// TIA Portal V18 export
VAR_GLOBAL   // PLC tag table "FactoryIO"
   "Emergency Stop 0" AT %I0.0 : Bool;
   "Start Button 0" AT %I0.1 : Bool;
   "Stop Button 0" AT %I0.2 : Bool;
   "Reset Button 0" AT %I0.3 : Bool;
   "Machining Center 0 (Is Busy)" AT %I0.5 : Bool;
   "Machining Center 0 (Has Error)" AT %I0.6 : Bool;
   "Machining Center 1 (Is Busy)" AT %I0.7 : Bool;
   "Machining Center 1 (Has Error)" AT %I1.0 : Bool;
   "Sensor 120" AT %I1.1 : Bool;
   "Sensor 122" AT %I1.2 : Bool;
   "Zne01 Conveyor 101" AT %Q0.0 : Bool;
   "Zne01 Conveyor 120" AT %Q0.1 : Bool;
   "Zne01 Conveyor 121" AT %Q0.2 : Bool;
   "Zne01 Conveyor 122" AT %Q0.3 : Bool;
   "Zne01 Conveyor 124" AT %Q0.4 : Bool;
   "Zne01 Conveyor 125" AT %Q0.5 : Bool;
   "Zne01 Sorter 102 (Up)" AT %Q0.6 : Bool;
   "Zne01 Sorter 102 (Left)" AT %Q0.7 : Bool;
   "Zne01 Sorter 102 (Right)" AT %Q1.0 : Bool;
   "Zne01 Sorter 123 (Up)" AT %Q1.1 : Bool;
   "Zne01 Sorter 123 (Right)" AT %Q1.2 : Bool;
   "Machining Center 0 (Start)" AT %Q1.3 : Bool;
   "Machining Center 0 (Stop)" AT %Q1.4 : Bool;
   "Machining Center 0 (Reset)" AT %Q1.5 : Bool;
   "Machining Center 1 (Start)" AT %Q1.6 : Bool;
   "Machining Center 1 (Stop)" AT %Q1.7 : Bool;
   "Machining Center 1 (Reset)" AT %Q2.0 : Bool;
   "Start Button 0 (Light)" AT %Q2.1 : Bool;
   "Stop Button 0 (Light)" AT %Q2.2 : Bool;
   "Reset Button 0 (Light)" AT %Q2.3 : Bool;
   "Vision Sensor 0 (Value)" AT %IW256 : Int;
   "Auto Selector 0" AT %I0.4 : Bool;
   "Machining Center 2 (Is Busy)" AT %I1.3 : Bool;
   "Machining Center 2 (Has Error)" AT %I1.4 : Bool;
   "Machining Center 3 (Is Busy)" AT %I1.5 : Bool;
   "Machining Center 3 (Has Error)" AT %I1.6 : Bool;
   "Sensor 130" AT %I1.7 : Bool;
   "Sensor 132" AT %I2.0 : Bool;
   "Zne01 Conveyor 130" AT %Q2.4 : Bool;
   "Zne01 Conveyor 131" AT %Q2.5 : Bool;
   "Zne01 Conveyor 132" AT %Q2.6 : Bool;
   "Zne01 Conveyor 134" AT %Q2.7 : Bool;
   "Zne01 Conveyor 135" AT %Q3.0 : Bool;
   "Zne01 Sorter 133 (Up)" AT %Q3.1 : Bool;
   "Zne01 Sorter 133 (Left)" AT %Q3.2 : Bool;
   "Machining Center 2 (Start)" AT %Q3.3 : Bool;
   "Machining Center 2 (Stop)" AT %Q3.4 : Bool;
   "Machining Center 2 (Reset)" AT %Q3.5 : Bool;
   "Machining Center 3 (Start)" AT %Q3.6 : Bool;
   "Machining Center 3 (Stop)" AT %Q3.7 : Bool;
   "Machining Center 3 (Reset)" AT %Q4.0 : Bool;
   "Zne02 Conveyor 220" AT %Q4.1 : Bool;
   "Zne02 Conveyor 221" AT %Q4.2 : Bool;
   "Zne02 Conveyor 222A" AT %Q4.3 : Bool;
   "Zne02 Conveyor 222B" AT %Q4.4 : Bool;
   "Zne02 Conveyor 223" AT %Q4.5 : Bool;
   "Zne02 Conveyor 224" AT %Q4.6 : Bool;
   "Zne02 Conveyor 225" AT %Q4.7 : Bool;
   "Zne03 Conveyor 300" AT %Q5.3 : Bool;
   "Zne03 Conveyor 301" AT %Q5.4 : Bool;
   "Zne03 Conveyor 302" AT %Q5.5 : Bool;
   "Sensor 223" AT %I2.1 : Bool;
   "Sensor 225" AT %I2.2 : Bool;
   "Zne02 Clamp Closed" AT %I2.3 : Bool;
   "Zne02 Clamp Limit" AT %I2.4 : Bool;
   "Zne02 Pusher" AT %Q5.0 : Bool;
   "Zne02 Clamp" AT %Q5.1 : Bool;
   "Zne02 Clamp Rise" AT %Q5.2 : Bool;
   "Vision Sensor 2 (Value)" AT %IW258 : Int;
   "Sensor 300" AT %I2.5 : Bool;
   "Sensor 301" AT %I2.6 : Bool;
   "Sensor 302" AT %I2.7 : Bool;
   "Zne03 (Detected)" AT %I3.0 : Bool;
   "Zne03 (Moving X)" AT %I3.1 : Bool;
   "Zne03 (Moving Z)" AT %I3.2 : Bool;
   "Zne03 Clamp Closed" AT %I3.3 : Bool;
   "Zne03 Clamp Limit" AT %I3.4 : Bool;
   "Zne03 Clamp" AT %Q5.6 : Bool;
   "Zne03 Clamp Raise" AT %Q5.7 : Bool;
   "Zne03 X" AT %Q6.0 : Bool;
   "Zne03 Z" AT %Q6.1 : Bool;
   "Zne03 (Grab)" AT %Q6.2 : Bool;
   "Zne03 Pusher" AT %Q6.3 : Bool;
   "Vision Sensor 1 (Value)" AT %IW260 : Int;
   "Sensor 423" AT %I3.5 : Bool;
   "Sensor 425" AT %I3.6 : Bool;
   "Zne04 Clamp Closed" AT %I3.7 : Bool;
   "Zne04 Clamp Limit" AT %I4.0 : Bool;
   "Sensor 500" AT %I4.1 : Bool;
   "Sensor 501" AT %I4.2 : Bool;
   "Sensor 502" AT %I4.3 : Bool;
   "Zne05 (Detected)" AT %I4.4 : Bool;
   "Zne05 (Moving X)" AT %I4.5 : Bool;
   "Zne05 (Moving Z)" AT %I4.6 : Bool;
   "Zne05 Clamp Closed" AT %I4.7 : Bool;
   "Zne05 Clamp Limit" AT %I5.0 : Bool;
   "Zne04 Conveyor 420" AT %Q6.4 : Bool;
   "Zne04 Conveyor 421" AT %Q6.5 : Bool;
   "Zne04 Conveyor 422B" AT %Q6.7 : Bool;
   "Zne04 Conveyor 423" AT %Q7.0 : Bool;
   "Zne04 Conveyor 424" AT %Q7.1 : Bool;
   "Zne04 Conveyor 425" AT %Q7.2 : Bool;
   "Zne04 Pusher" AT %Q7.3 : Bool;
   "Zne04 Clamp" AT %Q7.4 : Bool;
   "Zne04 Clamp Raise" AT %Q7.5 : Bool;
   "Zne05 Conveyor 500" AT %Q7.6 : Bool;
   "Zne05 Conveyor 501" AT %Q7.7 : Bool;
   "Zne05 Conveyor 502" AT %Q8.0 : Bool;
   "Zne05 Clamp" AT %Q8.1 : Bool;
   "Zne05 Clamp Raise" AT %Q8.2 : Bool;
   "Zne05 X" AT %Q8.3 : Bool;
   "Zne05 Z" AT %Q8.4 : Bool;
   "Zne05 (Grab)" AT %Q8.5 : Bool;
   "Zne05 Pusher" AT %Q8.6 : Bool;
   "Vision Sensor 3 (Value)" AT %IW262 : Int;
   "Vision Sensor 4 (Value)" AT %IW264 : Int;
   "Zne04 Conveyor 422A" AT %Q6.6 : Bool;
   "Sensor 920" AT %I10.0 : Bool;
   "Sensor 921" AT %I10.1 : Bool;
   "Sensor 922" AT %I10.2 : Bool;
   "Sensor 930" AT %I10.3 : Bool;
   "Sensor 931" AT %I10.4 : Bool;
   "Sensor 932" AT %I10.5 : Bool;
   "Sensor 950" AT %I10.6 : Bool;
   "Sensor 951" AT %I10.7 : Bool;
   "Sensor 952" AT %I11.0 : Bool;
   "Sensor 953" AT %I11.1 : Bool;
   "Zne09 Conveyor 920" AT %Q10.0 : Bool;
   "Zne09 Conveyor 921" AT %Q10.1 : Bool;
   "Zne09 Conveyor 930" AT %Q10.2 : Bool;
   "Zne09 Conveyor 931" AT %Q10.3 : Bool;
   "Zne09 Conveyor 950" AT %Q10.4 : Bool;
   "Zne09 Conveyor 951" AT %Q10.5 : Bool;
   "Zne09 Conveyor 952" AT %Q10.6 : Bool;
   "Zne09 Conveyor 953" AT %Q10.7 : Bool;
   "Zne09 Chain Transfer Right" AT %Q11.0 : Bool;
   "Zne09 Chain Transfer Left" AT %Q11.1 : Bool;
   "Zne09 Chain Transfer Foward" AT %Q11.2 : Bool;
   "Zne09 Chain Transfer Backward" AT %Q11.3 : Bool;
   "Pick & Place 0 X Position (V)" AT %IW266 : Int;
   "Pick & Place 0 Y Position (V)" AT %IW268 : Int;
   "Pick & Place 0 Z Position (V)" AT %IW270 : Int;
   "Pick & Place 1 X Position (V)" AT %IW272 : Int;
   "Pick & Place 1 Y Position (V)" AT %IW274 : Int;
   "Pick & Place 1 Z Position (V)" AT %IW276 : Int;
   "Pick & Place 0 X Set Point (V)" AT %QW256 : Int;
   "Pick & Place 0 Y Set Point(V)" AT %QW258 : Int;
   "Pick & Place 0 Z Set Point (V)" AT %QW260 : Int;
   "Pick & Place 1 X Set Point (V)" AT %QW262 : Int;
   "Pick & Place 1 Y Set Point(V)" AT %QW264 : Int;
   "Pick & Place 1 Z Set Point (V)" AT %QW266 : Int;
   "Zne09 Stacker Target Position" AT %QW270 : Int;
   "Pick & Place 1 (Box Detected)" AT %I11.2 : Bool;
   "Pick & Place 0 (Box Detected)" AT %I11.3 : Bool;
   "Pick & Place 1 (Grab)" AT %Q11.4 : Bool;
   "Pick & Place 0 (Grab)" AT %Q11.5 : Bool;
   AtRight AT %I12.0 : Bool;
   AtLeft AT %I12.1 : Bool;
   AtCenter AT %I12.2 : Bool;
   MovingX AT %I12.3 : Bool;
   MovingZ AT %I12.4 : Bool;
   "Forks RIght" AT %Q12.0 : Bool;
   ForksLeft AT %Q12.1 : Bool;
   Lift AT %Q12.2 : Bool;
END_VAR
VAR_GLOBAL CONSTANT   // user constants
   BlueRawMaterial : Int := 1;
   GreenRawMaterial : Int := 4;
   HOMEPOSITION : Int := 255;
   BlueLidMaterial : Int := 2;
   GreenLidMaterial : Int := 5;
   BlueBaseMaterial : Int := 3;
   GreenBaseMaterial : Int := 6;
   MaxCoordinates : Int := 10;
END_VAR
